FUNCTION_BLOCK LIFT
VAR_INPUT
	LiftRun : BOOL;
	DOOR_OPEN : BOOL;    //
	RaklapInLift : BOOL; // I 0.6
	
	
	//PalettLoaded : BOOL;
END_VAR
VAR_OUTPUT
	LiftUp : BOOL;
	LiftDown : BOOL;
	LiftEnd : BOOL;
	LiftReady : BOOL;
	LiftPos : INT;	
	Raklap_IN : BOOL; //Raklap be szalag 
	Raklap_OUT :BOOL; //Raklap ki szalag
	
END_VAR



VAR
CaseN : INT;	
F_Ready : F_TRIG;
LayerCount : INT;
Open_TIME : TON;
PUSH_OUT : TON;

END_VAR





PUSH_OUT(IN:= Raklap_OUT, PT := T#3S);


Open_TIME(IN:=DOOR_OPEN, PT:= T#4S);


IF Open_TIME.Q THEN
	LayerCount := LayerCount + 1;
END_IF


CASE CaseN OF

	
0:
		Raklap_IN := 1;
		
	IF RaklapInLift THEN 
	Raklap_IN := 0;   // Raklap bent
		CaseN := 20;
	
	END_IF
20:							//lift felmegy
		LiftUp := 1;
		LiftEnd := 1;
		LayerCount := 0;   //Layer reset
	IF LiftRun = 0 THEN
		CaseN := 30;
		LiftPos := 0;
	
	END_IF
30:						//Lift lemegy egy lépést
	LiftDown:= 1;
	CaseN:= 31;
	
	
31:
LiftDown := 0;
IF LiftRun = 0 THEN
LiftReady := 1;
LiftPos := 1;
CaseN := 40;
END_IF


40:
	
IF LayerCount = 1 THEN   // első sor megvan le mozog a lift
	LiftDown := 1;
	LiftReady := 0;
	
	CaseN := 41;
	END_IF
41:
LiftDown := 0;
IF LiftRun = 0 THEN     
LiftReady := 1;
LiftPos := 2;
CaseN := 40;
END_IF


50: 

IF LayerCount = 2 THEN   // második sor megvan le mozog a lift
	LiftDown := 1;
	LiftReady := 0;
	
	CaseN := 51;
	END_IF
51:
LiftDown := 0;
IF LiftRun = 0 THEN     
LiftReady := 1;
LiftPos := 3;
CaseN := 60;
END_IF

60: 

IF LayerCount = 2 THEN   // Harmadik sor megvan le mozog a lift végállásig
	LiftDown := 1;
	LiftEnd := 1;
	LiftReady := 0;
	
	CaseN := 61;
	END_IF
61:

IF LiftRun = 0 THEN      
LiftPos := 4;
LiftDown := 0;
LiftEnd := 0;
CaseN := 70;
END_IF
	
70:										//Lift kirakod
	Raklap_OUT := 1;
	CaseN := 71;
	
71:
	IF PUSH_OUT.Q = 1 THEN
		Raklap_OUT := 0;
		CaseN := 0;
	END_IF


END_CASE

END_FUNCTION_BLOCK

(* stored: Version 1.1.0.1, ProductVersion 3.1.4024.11
   POU LIFT: Id {fe2b07cc-ed9f-4fb9-8a70-1b754d8ab060}, SpecialFunc None *)
